PROGRAM PRG_00_General
VAR
	sr_Fault: SR;
	FB_Blinker_ServoError: FB_Blinker;
	FB_Blinker_RetainError: FB_Blinker;
END_VAR
VAR // added by the converter: edge detectors and wires of the graphical bodies
    _w1 : BOOL;
END_VAR

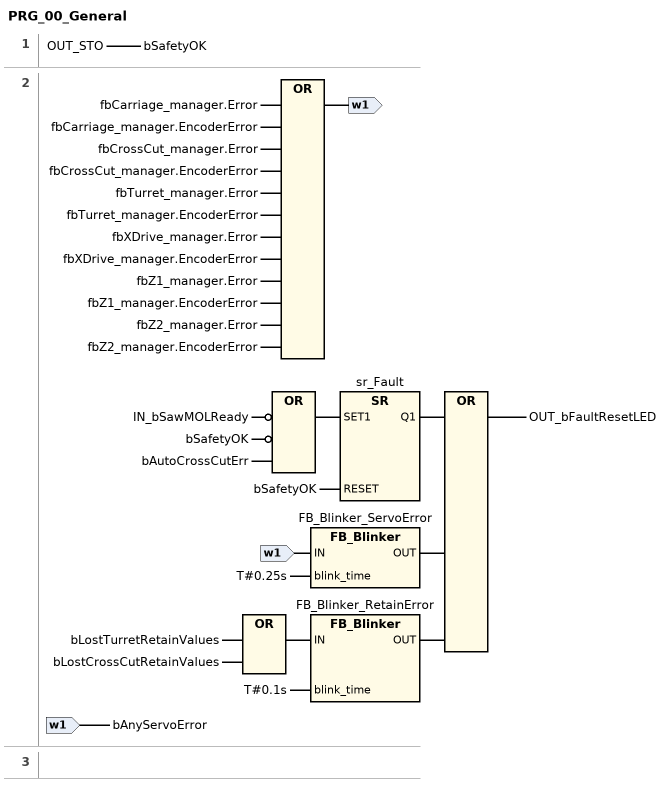
// NETWORK 1
bSafetyOK := OUT_STO;

// NETWORK 2
_w1 := fbCarriage_manager.Error OR fbCarriage_manager.EncoderError OR fbCrossCut_manager.Error OR fbCrossCut_manager.EncoderError OR fbTurret_manager.Error OR fbTurret_manager.EncoderError OR fbXDrive_manager.Error OR fbXDrive_manager.EncoderError OR fbZ1_manager.Error OR fbZ1_manager.EncoderError OR fbZ2_manager.Error OR fbZ2_manager.EncoderError;
sr_Fault(SET1 := NOT IN_bSawMOLReady OR NOT bSafetyOK OR bAutoCrossCutErr, RESET := bSafetyOK); // SR
FB_Blinker_ServoError(IN := _w1, blink_time := T#0.25s); // FB_Blinker
FB_Blinker_RetainError(IN := bLostTurretRetainValues OR bLostCrossCutRetainValues, blink_time := T#0.1s); // FB_Blinker
OUT_bFaultResetLED := sr_Fault.Q1 OR FB_Blinker_ServoError.OUT OR FB_Blinker_RetainError.OUT;
bAnyServoError := _w1;

// NETWORK 3

END_PROGRAM

(* stored: Version 1.1.0.1, ProductVersion 3.1.4024.15
   POU PRG_00_General: Id {e2f2a1d5-cf74-4250-a3bf-c8c0897f0dd8}, SpecialFunc None *)
